// TwinCAT 3 PLC project CompA_TCP_Server
// ProgramVersion: 3.1.0.5
// libraries:
//   Tc2_Standard, * (Beckhoff Automation GmbH)
//   Tc2_System, * (Beckhoff Automation GmbH)
//   Tc2_TcpIp, * (Beckhoff Automation GmbH)
//   Tc2_Utilities, * (Beckhoff Automation GmbH)
//   Tc3_Module, * (Beckhoff Automation GmbH)
// project tree:
//   Data types/ ST_ApplicationBinaryData.TcDUT, ST_BinaryFrame.TcDUT (not stored), ST_BinaryHeader.TcDUT
//   Global Variables/ Global_Variables.TcGVL (not stored)
//   / PlcTaskServer.TcTTO (not stored)
//   POUs/ FB_Server.TcPOU (not stored), FB_ServerApplication.TcPOU, FB_ServerConnection.TcPOU (not stored), MAIN.TcPOU
//   POUs/Helper POUs/ FB_FrameFifo.TcPOU (not stored), FB_LogFifo.TcPOU (not stored), F_ADSLOGHEXDATA.TcPOU (not stored)
// real-time tasks:
//   TASK PlcTaskServer: cycle T#10ms, priority 21, ADS port 351

// ---- Data types/ST_ApplicationBinaryData.TcDUT
(* Simple binary user data (8 byte aligned) *)
TYPE ST_ApplicationBinaryData :
STRUCT
	fPos		:  LREAL;(* 8 byte *)
END_STRUCT
END_TYPE

// ---- Data types/ST_BinaryHeader.TcDUT
(* Simple binary TCP/IP frame header (8 byte aligned) *)
TYPE ST_BinaryHeader :
STRUCT
	dwStart		: DWORD	:= 16#BECF1234;	(* Start bytes *)
	cbLength	: UDINT(0..PLCPRJ_BUFFER_SIZE) := 0;(* Max. length of attached binary data *)
	nS			: UDINT := 0;(* Send counter *)
	nR			: UDINT	:= 0;(* Receive counter *)
	
	
	(* Total header data size = 16 byte *)
END_STRUCT
END_TYPE

// ---- POUs/FB_ServerApplication.TcPOU
(* Comp A TCP Server*)
FUNCTION_BLOCK FB_ServerApplication
VAR_IN_OUT
	fbTx 			: FB_FrameFifo;(* TX fifo *)
	fbRx 			: FB_FrameFifo;(* RX fifo *)
	fbLog			: FB_LogFifo;(* Log message fifo *)
END_VAR
VAR
	stToClient		: ST_ApplicationBinaryData; (* Tx user data *)
	stFromClient	: ST_ApplicationBinaryData; (* Rx user data *)
	stTxFrame		: ST_BinaryFrame;(* Tx frame buffer (inclusive header) *)
	stRxFrame		: ST_BinaryFrame;(* Rx frame buffer (inclusive header) *)
	state: INT := 0;
	CompBData: LREAL;(* 8 byte *)
	nStateTPC: INT := 0;
END_VAR
VAR PERSISTENT
	ToggleCount: INT := 0;
END_VAR
VAR CONSTANT
	nToogleCycle: INT := 5;
END_VAR

REPEAT		
	(*TPC States* - State Machine Implementation*)	
	CASE nStateTPC OF
	0:(* CLOSED STATE *)
	    stFromClient := fbRx.stGet;  (*RECEIVE SYN*)
		IF ( stFromClient.fpos  <> 0) THEN
			stFromClient.fpos :=HEXSTR_TO_DATA('000007D0', ADR( stFromClient.fpos ), SIZEOF( stFromClient.fpos ) ); (* SEND SYN -ACK*)
			fbTx.AddTail( stPut := stToClient );
			stFromClient.fpos := HEXSTR_TO_DATA('000003E9', ADR( stFromClient.fpos ), SIZEOF( stFromClient.fpos ) );
			fbTx.AddTail( stPut := stToClient );			
			state:=1;
		ELSE
			state:=0;
		END_IF
		
	1: (* SYN RECEIVED STATE*)
		stFromClient := fbRx.stGet;
		IF (stFromClient.fpos =  HEXSTR_TO_DATA('000007D1', ADR( stFromClient.fpos ), SIZEOF( stFromClient.fpos ) )) THEN (*RECEIVED ACK *)
			state:=2;
		ELSE
			state:=1;
		END_IF
		
	2: (* ESTABLISHED STATE*)
		 (* Toogle server data every 5*100 ms*)
		 IF(ToggleCount< nToogleCycle) THEN
			stToClient.fpos:=HEXSTR_TO_DATA('88888888', ADR( stFromClient.fpos ), SIZEOF( stFromClient.fpos ) );  
			ToggleCount := ToggleCount +1 ;
		 ELSE
			stToClient.fpos:=HEXSTR_TO_DATA('88888889', ADR( stFromClient.fpos ), SIZEOF( stFromClient.fpos ) );
			ToggleCount := 0;
		 END_IF
		 fbTx.AddTail( stPut := stToClient ); (* send CompA server data*)
		 stFromClient := fbRx.stGet; (* received ACK*)
		 IF ( stFromClient.fpos = HEXSTR_TO_DATA('000007D1', ADR( stFromClient.fpos ), SIZEOF( stFromClient.fpos ) ) ) THEN
			 stFromClient := fbRx.stGet; (* get CompB Client data*)
			 IF ( stFromClient.fpos <> 0 )THEN 
                CompBData :=  stFromClient.fpos;   
				stToClient.fpos :=  HEXSTR_TO_DATA('000007D1', ADR( stFromClient.fpos ), SIZEOF( stFromClient.fpos ) ); (*send ACK*)
				fbTx.AddTail( stPut := stToClient );
			 END_IF
		  END_IF
		  
		  stFromClient := fbRx.stGet; (* received FIN*)	  
		  IF ( stFromClient.fpos=  HEXSTR_TO_DATA('000003E8', ADR( stFromClient.fpos ), SIZEOF( stFromClient.fpos ) ) )THEN    (* send ACK for client data *)
				stToClient.fpos :=  HEXSTR_TO_DATA('000003E9', ADR( stFromClient.fpos ), SIZEOF( stFromClient.fpos ) );
				fbTx.AddTail( stPut := stToClient );
				state:=3;
		  ELSE
			  state:=2;
		  END_IF
	
	3:  (* CLOSE WAIT STATE*)
		 stToClient.fpos := HEXSTR_TO_DATA('000003E9', ADR( stFromClient.fpos ), SIZEOF( stFromClient.fpos ) );   (* send FIN  for close *)
		 fbTx.AddTail( stPut := stToClient );
		 state :=4;
	
	
	4:  (* LAST ACK STATE*)
		 stFromClient := fbRx.stGet;
		 IF (stFromClient.fpos = HEXSTR_TO_DATA('000005BF', ADR( stFromClient.fpos ), SIZEOF( stFromClient.fpos ) ) ) THEN
			state:=0;	 
		 END_IF
	
	END_CASE
	
UNTIL NOT fbRx.bOk
END_REPEAT

END_FUNCTION_BLOCK

// ---- POUs/MAIN.TcPOU
PROGRAM MAIN
VAR
	sSrvNetID		: T_AmsNetID	:= '';(* TwinCAT TCP/IP server network address *)
	sLocalHost		: T_Ipv4Addr 	:= '127.0.0.1';(* Server IP network address *)
	nLocalPort		: UDINT 		:= 200;(* Server port number *)
	bEnable			: BOOL 			:= TRUE;(* TRUE => Enable server data exchange, FALSE => Disable *)
	bLog			: BOOL			:= TRUE;(* TRUE => Enable log message output, FALSE => Disable *)
	fbServer		: FB_Server := ( sPrefix := 'SERVER::' );(* Server (connection) instance *)
	hServer			: T_HSERVER;(* Server connection handle *)

	fbCloseAll		: FB_SocketCloseAll;
	bInitialize		: BOOL := TRUE;
END_VAR

(* On PLC reset or program download close all old (opened) connections *)
fbCloseAll( sSrvNetID := sSrvNetID, bExecute:= bInitialize );
IF fbCloseAll.bBusy OR fbCloseAll.bError THEN
	RETURN;
END_IF

IF bInitialize THEN
	bInitialize := FALSE;

	(* Initialize server handle *)
	F_CreateServerHnd( 	sSrvNetID 	:= sSrvNetID,
						sLocalHost 	:= sLocalHost,
						nLocalPort	:= nLocalPort,
						nMode 		:= SEL( bLog, 0, CONNECT_MODE_ENABLEDBG ),(* Enable debug messages *)
						bEnable 	:= FALSE,(* TRUE = leave listener socket open, FALSE = close listener socket after last connection ist closed too *)
						hServer 	:= hServer );
END_IF


(* Trigger the execution of every server (connection) instance *)
fbServer( hServer := hServer, sSrvNetID := sSrvNetID, bEnable := bEnable, bLog := bLog );

END_PROGRAM
